% RSLogix 500 project P5_ASHLEY_J.RSS, saved by version 8.30.00.16 %
PROJECT "UNTITLED"    % processor: Bul.1763 MicroLogix 1100 Series B %

PROGRAM FILES
  LAD 2 "MAIN"  2 rungs
  LAD 3 "ROTAMETER"  6 rungs

DATA FILES
  O0 OUTPUT  4 elements
  I1 INPUT  6 elements
  S2 STATUS  66 elements
  B3 BINARY  1 elements
  T4 TIMER  2 elements
  C5 COUNTER  1 elements
  R6 CONTROL  1 elements
  N7 INTEGER  1 elements
  F8 FLOAT  4 elements

LADDER 2 "MAIN"
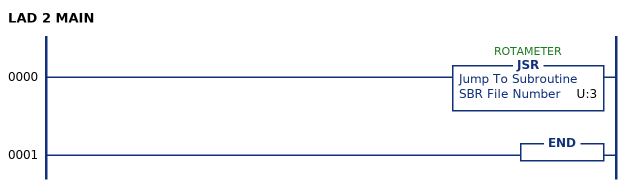
% Rung: 0 %
SOR JSR U:3 EOR
%   U:3  "ROTAMETER" %
% Rung: 1 %
SOR END EOR

LADDER 3 "ROTAMETER"
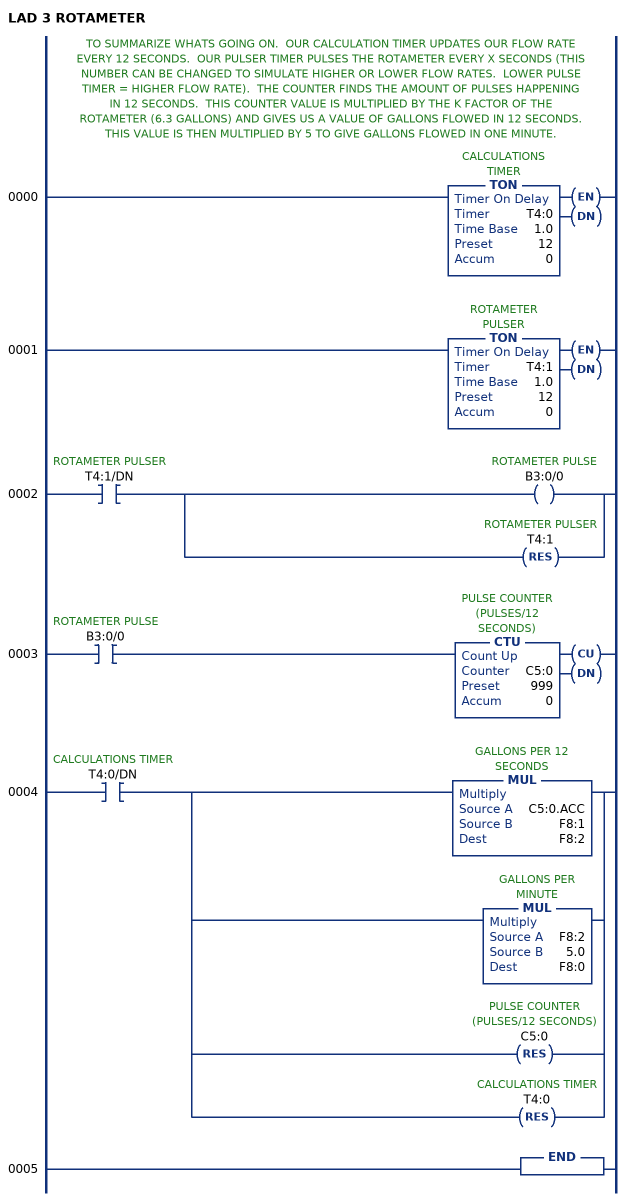
% Rung: 0 %
% TO SUMMARIZE WHATS GOING ON.  OUR CALCULATION TIMER UPDATES OUR FLOW RATE EVERY 12 SECONDS.  OUR PULSER TIMER PULSES THE ROTAMETER EVERY X SECONDS (THIS NUMBER CAN BE CHANGED TO SIMULATE HIGHER OR LOWER FLOW RATES.  LOWER PULSE TIMER = HIGHER FLOW RATE).  THE COUNTER FINDS THE AMOUNT OF PULSES HAPPENING IN 12 SECONDS.  THIS COUNTER VALUE IS MULTIPLIED BY THE K FACTOR OF THE ROTAMETER (6.3 GALLONS) AND GIVES US A VALUE OF GALLONS FLOWED IN 12 SECONDS.  THIS VALUE IS THEN MULTIPLIED BY 5 TO GIVE GALLONS FLOWED IN ONE MINUTE. %
SOR TON T4:0 1.0 12 0 EOR
%   T4:0  "CALCULATIONS TIMER" %
% Rung: 1 %
SOR TON T4:1 1.0 12 0 EOR
%   T4:1  "ROTAMETER PULSER" %
% Rung: 2 %
SOR XIC T4:1/DN BST OTE B3:0/0 NXB RES T4:1 BND EOR
%   T4:1  "ROTAMETER PULSER" %
%   B3:0/0  "ROTAMETER PULSE" %
% Rung: 3 %
SOR XIC B3:0/0 CTU C5:0 999 0 EOR
%   B3:0/0  "ROTAMETER PULSE" %
%   C5:0  "PULSE COUNTER (PULSES/12 SECONDS)" %
% Rung: 4 %
SOR XIC T4:0/DN BST MUL C5:0.ACC F8:1 F8:2 NXB MUL F8:2 5.0 F8:0 NXB RES C5:0 NXB RES T4:0 BND EOR
%   T4:0  "CALCULATIONS TIMER" %
%   C5:0  "PULSE COUNTER (PULSES/12 SECONDS)" %
%   F8:1  "K FACTOR (GALLONS PER PULSE)" %
%   F8:2  "GALLONS PER 12 SECONDS" %
%   F8:0  "GALLONS PER MINUTE" %
% Rung: 5 %
SOR END EOR

DATA TABLE (non-zero values as saved)
DATA T4
% .PRE .ACC %
% T4:0 % 12 0
% T4:1 % 12 0
DATA C5
% .PRE .ACC %
% C5:0 % 999 0
DATA F8
% F8:0 % 0 6.3 0 0
